INTERFACE ITF_Regelschuif_OutOpen_DG

METHOD set : BOOL
VAR_INPUT
	state : BOOL;
END_VAR
END_METHOD

END_INTERFACE

(* stored: Version 1.1.0.1, ProductVersion 3.1.4026.8
   Itf ITF_Regelschuif_OutOpen_DG: Id {55db5129-1bf3-45ba-8ec7-bda156a365aa}
   Method set: Id {ebabf594-8bc8-4d66-ac26-c10c8dc13dc6} *)
